// Mitsubishi GX Works2 project: 24   PLC: FX3G

// task Task_01 (event TRUE, interval 0, priority 31): POU_01

PROGRAM POU_01
VAR
  gas : INT;
  ton1 : TON;
  gas1 : INT;
  ton2 : TON;
END_VAR
IF M8002 THEN
gas := 0;
gas1:=0;
END_IF;
IF M2 THEN 
	gas1:=1;
	END_IF;

CASE gas OF
	0:
	Y0:=FALSE;
	Y1:=FALSE;
	Y2:=FALSE;
	Y3:=FALSE;
	IF M1 THEN
		gas:=1;
	END_IF;

	1:
	Y0:=TRUE;
	ton1(IN := NOT ton1.Q, PT := T#0.5s);
IF ton1.Q THEN
	gas:=2;
	Y0:=FALSE;
END_IF;

2:
Y1:=TRUE;
ton1(IN := NOT ton1.Q, PT := T#0.5s);
IF ton1.Q THEN
	gas:=3;
	Y1:=FALSE;
END_IF;

	3:
	Y2:=TRUE;
	ton1(IN := NOT ton1.Q, PT := T#0.5s);
IF ton1.Q THEN
	gas:=1;
	Y2:=FALSE;
END_IF;
END_CASE;

CASE gas1 OF
	1:
	Y3:=TRUE;
	ton2(IN := NOT ton2.Q, PT := T#5s);
IF ton2.Q THEN
	gas:=0;
	gas1:=0;
END_IF;
	
	END_CASE;
END_PROGRAM
